KUKA KRL data list: ConfGarra.dat

&ACCESS RVO1
&PARAM EDITMASK = *
DEFDAT ConfGarra

ENDDAT
